TYPE User1_Par :
STRUCT
 	// iTargetTorque	                 	:ARRAY[1..3]OF INT:= [3(-50)];			                     (*单位为0.1%*)
     iTest                                   :INT;

     parFilterAD              :ARRAY[1..MaxAINo] OF ST_ParFilterAD;
     parDA                     :ARRAY[1..44] OF INT;   //模拟量输出
	HMI_Version					:STRING:='V20221208';//触摸屏版本号
	PLC_Version					:STRING:='V20221208';//PLC版本号
    bSyncMode:INT:=1;//0=不同步启动叠台主轴，1=同时启动叠台主轴






END_STRUCT
END_TYPE

(* stored: Version 1.1.0.1, ProductVersion 3.1.4024.12
   DUT User1_Par: Id {cd9e9202-ea8c-4628-a757-038eeac69993} *)
